Fanuc KAREL source: kb00099.compact.KL

PROGRAM KB00099
%STACKSIZE=65535
%PRIORITY=65535
%NOLOCKGROUP
VAR
P1 : STRING[80]
P2 : STRING[80]
RESULT : INTEGER
BEGIN
P1='A'
P2='A'
RESULT=INDEX(P1,P2)
END KB00099
